FUNCTION_BLOCK TimeConvertor
VAR_INPUT
END_VAR
VAR_OUTPUT
END_VAR
VAR
END_VAR

METHOD fromfiletime64 : ST_TimeConvertor
VAR_INPUT
END_VAR
END_METHOD

END_FUNCTION_BLOCK

(* stored: Version 1.1.0.1, ProductVersion 3.1.4024.12
   POU TimeConvertor: Id {e1ad951e-bed6-4619-bb16-78dcbf2fd0cf}, SpecialFunc None
   Method fromfiletime64: Id {40514550-2e7d-4dac-83e9-9550db830ce5} *)
